# B&R Automation Studio project PloterCNC (part 6)

#### Main.st
```iecst
PROGRAM _INIT
	gParameter;
	UISetup.RecipeListSize	:= 20;
	i; // selected index

END_PROGRAM

PROGRAM _CYCLIC

	// basic settings for recipes
	MpRecipeXml_0(MpLink := ADR(gRecipeXml), Enable := TRUE, DeviceName := ADR('CF'), FileName := ADR('recipe') );

	MpRecipeRegPar_0(MpLink := ADR(gRecipeXml), Enable := TRUE, PVName := ADR('gParameter') );

	MpRecipeUI_0(MpLink := ADR(gRecipeXml), Enable := TRUE, UISetup := UISetup, UIConnect := ADR(UIConnect));

	UIConnect.Recipe.Filter:='*.xml';

	FOR k:=0 TO 4 DO
		memset(ADR(TempLine[k]),0,SIZEOF(TempLine[k]));
		memset(ADR(DataProvider0[k]),0, SIZEOF(DataProvider0[k]));
	END_FOR;

	FOR i:=0 TO 4 DO
		TempLine[0]:='{"value":"';
		TempLine[1]:=INT_TO_STRING(i);
		TempLine[2]:='","text":"';
		TempLine[3]:=UIConnect.Recipe.List.Names[i];
		TempLine[4]:='"}';

		nextAddr:=strcat(ADR(DataProvider0[i]), ADR(TempLine[0]));

		FOR j:=1 TO 4 DO
			strcat(nextAddr,ADR(TempLine[j]));
		END_FOR;

	END_FOR;

	// Messagebox informs that the maximum number of recipes has been reached

	IF UIConnect.Recipe.List.MaxSelection>=5 AND CreatingRecipe  THEN
		gMsgBox4:=TRUE;
		CreatingRecipe := FALSE;
	END_IF;

		END_PROGRAM

PROGRAM _EXIT

	MpRecipeXml_0.Save					:= TRUE;
	MpRecipeXml_0.Enable				:=FALSE;
	MpRecipeXml_0();

	MpRecipeRegPar_0.Enable				:=FALSE;
	MpRecipeRegPar_0();

		END_PROGRAM
```

### Program Logical/RuchZGCode

#### Main.st
```iecst
PROGRAM _INIT
	(* Insert code here *)
	CncName := '';
	CncNameCopy := '';
	toolDown;
	toolUp;
	MC_BR_MFunction_0(AxesGroup :=ADR(gCncXZ) , Enable :=TRUE , MFunction :=50);
	MC_BR_MFunction_1(AxesGroup :=ADR(gCncXZ) , Enable :=TRUE , MFunction :=60);
END_PROGRAM

PROGRAM _CYCLIC

	//Transfering name of the opened file in MotionPad to the initialization of CNC

	IF MpCnc2Axis_0.PowerOn AND MpCnc2Axis_0.IsHomed AND MoveMachine = 1 THEN

	CncNameCopy := DELETE(CncName, 12, 0);
		CncParameters.ProgramName := CncNameCopy;
		MoveMachine := 2;
		IF  strcmp(ADR(CncNameCopy),ADR('')) <> 0 THEN
			MpCnc2Axis_0.MoveProgram := TRUE;
		END_IF

	ELSIF MpCnc2Axis_0.MoveDone THEN
		CncName := '';
		CncNameCopy := '';
		MpCnc2Axis_0.MoveProgram := FALSE;
	END_IF

	//Error control, showing the Error Dialog and reseting errors
	IF MpCnc2Axis_0.Error THEN
		DialogErrorVisible := TRUE;
		MpCnc2Axis_0.Stop := TRUE;
		MpCnc2Axis_0.MoveProgram := FALSE;
	END_IF

	IF MpCnc2Axis_0.Error = FALSE THEN
		MpCnc2Axis_0.ErrorReset := FALSE;
	END_IF

	MC_BR_MFunction_0();
	MC_BR_MFunction_1();
	IF EDGEPOS(toolUp) THEN
		gActiveTool:=FALSE;
		MC_BR_MFunction_0.Reset:=TRUE;
	ELSE
		MC_BR_MFunction_0.Reset:=FALSE;
	END_IF

	IF EDGEPOS(toolDown) THEN
		gActiveTool:=TRUE;
		MC_BR_MFunction_1.Reset:=TRUE;
	ELSE
		MC_BR_MFunction_1.Reset:=FALSE;
	END_IF

END_PROGRAM

PROGRAM _EXIT
	(* Insert code here *)

END_PROGRAM
```

### Package Logical/Sources/Infrastructure - Infrastructure package

### Program Logical/Sources/Infrastructure/SMTP (IEC) - Mail notification via smtp task

#### Smtp.st - Smtp init, cyclic, exit code
```iecst
(*********************************************************************************
 * Copyright:	Bernecker+Rainer
 * Author:		pawlikb
 * Created:		April 23, 2019/8:53 AM
 * Description:
 *			What:	Task handles e-mail notfications about active alarms.
 *			How:	Timer is counting up to INTERVAL_TIME. During this time active
					alarms are registered and then the e-mail with combined information is sent
					and the timer is reset.
 *			Limits:	It is necessary to provide Internet access for the PLC.
					When used with SiteManager the default gateway must be set to DEV IP of the SiteManager,
					and Routing (Scada) Agent must be configured. Please see attached documentation.

 *********************************************************************************)

PROGRAM _INIT
	(* Smtp default configuration *)
	Smtp.Parameters.Host		:=	HOST;
	Smtp.Parameters.User		:=	USER;
	Smtp.Parameters.Password	:=	PASSWORD;
	Smtp.Parameters.Sender		:=	SENDER;
	Smtp.Parameters.Receiver	:=	RECEIVER;
	Smtp.Parameters.Subject		:=	SUBJECT;
	Smtp.Parameters.Text		:=	HEADER;
	Smtp.Parameters.Domain		:=	DOMAIN;				//Usually domain name is not needed
	Smtp.Parameters.Timeout		:=	0;					//If 0 specified then default 120s is used
	Smtp.Parameters.Port		:=	PORT;				//If 0 specified then default port for SMTP (25) is used

	(* Attachment *)
	Smtp.Parameters.AttachmentCnt		:=	0;
	Smtp.Parameters.Attachment.type		:=	smtpATT_TYPE_DATMOD;
	Smtp.Parameters.Attachment.pData	:=	ADR('DatObj');

	(* Timer configuration - get task class cycle time *)
	Smtp.FB.RTInfo.enable	:=	TRUE;
	Smtp.FB.RTInfo();

END_PROGRAM

PROGRAM _CYCLIC

//	(* Increment timer *)
//	Smtp.Status.Timer	:=	Smtp.Status.Timer + Smtp.FB.RTInfo.cycle_time/1000;
//
//	(* Reset timer and send e-mail *)
//	IF Smtp.Status.Timer >= (INTERVAL_TIME * 60) THEN
//		Smtp.Status.Timer	:=	0;
//
//		(* Send email if any alarm was set *)
//		IF Smtp.Status.AlarmActive THEN
////			Smtp.Cmd.Send		:=	TRUE;
////			Smtp.Cmd.SendSSL	:=	TRUE;
//		END_IF;
//	END_IF;
//
//	(* Check for active alarms *)
//	Smtp.Status.AlarmActive	:=	FALSE;
//	FOR i:=0 TO 10 DO
////		Smtp.Status.AlarmActive	:=	Smtp.Status.AlarmActive	OR	[i];
//
//	END_FOR;

	(* Disable function blocks - will be enabled in a state machine *)
	Smtp.FB.SmtpSend.enable		:=	FALSE;
	Smtp.FB.SmtpsSend.enable	:=	FALSE;

	(* State machine *)
	CASE Smtp.Status.State OF

		STATE_SMTP_WAIT:
			(* Command send via SMTP *)
			IF Smtp.Cmd.Send THEN
				(* Prepare message *)
				actText;
				(* Send *)
				Smtp.Status.State	:=	STATE_SMTP_SEND;
			END_IF;

			(* Command send via SMTP with encryption *)
			IF Smtp.Cmd.SendSSL THEN
				(* Prepare message *)
				actText;
				(* Send *)
				Smtp.Status.State	:=	STATE_SMTP_SEND_SSL;
			END_IF;

		STATE_SMTP_SEND:
			(* Enable function block *)
			Smtp.FB.SmtpSend.enable	:=	TRUE;

			(* Assign Mail Parameters *)
			Smtp.FB.SmtpSend.pHost			:=	ADR(Smtp.Parameters.Host);
			Smtp.FB.SmtpSend.pUser			:=	0;	//ADR(Smtp.Parameters.User);
			Smtp.FB.SmtpSend.pPassword		:=	0;	//ADR(Smtp.Parameters.Password);
			Smtp.FB.SmtpSend.pSender		:=	ADR(Smtp.Parameters.Sender);
			Smtp.FB.SmtpSend.pReceiver		:=	ADR(Smtp.Parameters.Receiver);
			Smtp.FB.SmtpSend.pSubject		:=	ADR(Smtp.Parameters.Subject);
			Smtp.FB.SmtpSend.pText			:=	ADR(Smtp.Parameters.Text);
			Smtp.FB.SmtpSend.pDomain		:=	0;	//ADR(Smtp.Parameters.Domain);
			Smtp.FB.SmtpSend.pAttachment	:=	ADR(Smtp.Parameters.Attachment);
			Smtp.FB.SmtpSend.attcnt			:=	Smtp.Parameters.AttachmentCnt;
			Smtp.FB.SmtpSend.timeout		:=	Smtp.Parameters.Timeout;
			Smtp.FB.SmtpSend.port			:=	Smtp.Parameters.Port;

			(* Jump Conditions *)
			IF Smtp.FB.SmtpSend.status = ERR_OK THEN
				Smtp.FB.SmtpSend.enable	:=	FALSE;
				Smtp.Status.State		:=	STATE_SMTP_WAIT;
			ELSIF Smtp.FB.SmtpSend.status = ERR_FUB_BUSY THEN
				(* BUSY *)
			ELSE
				Smtp.Status.State	:=	STATE_SMTP_ERROR;
			END_IF;

		STATE_SMTP_SEND_SSL:
			(* Enable function block *)
			Smtp.FB.SmtpsSend.enable	:=	TRUE;

			(* Assign Mail Parameters *)
			Smtp.FB.SmtpsSend.pHost			:=	ADR(Smtp.Parameters.Host);
			Smtp.FB.SmtpsSend.pUser			:=	ADR(Smtp.Parameters.User);
			Smtp.FB.SmtpsSend.pPassword		:=	ADR(Smtp.Parameters.Password);
			Smtp.FB.SmtpsSend.pSender		:=	ADR(Smtp.Parameters.Sender);
			Smtp.FB.SmtpsSend.pReceiver		:=	ADR(Smtp.Parameters.Receiver);
			Smtp.FB.SmtpsSend.pSubject		:=	ADR(Smtp.Parameters.Subject);
			Smtp.FB.SmtpsSend.pText			:=	ADR(Smtp.Parameters.Text);
			Smtp.FB.SmtpsSend.pDomain		:=	ADR(Smtp.Parameters.Domain);
			Smtp.FB.SmtpsSend.pAttachment	:=	ADR(Smtp.Parameters.Attachment);
			Smtp.FB.SmtpsSend.attcnt		:=	Smtp.Parameters.AttachmentCnt;
			Smtp.FB.SmtpsSend.timeout		:=	Smtp.Parameters.Timeout;
			Smtp.FB.SmtpsSend.port			:=	Smtp.Parameters.Port;
			Smtp.FB.SmtpsSend.sslCfgIdent	:=	0;	//Default SSL Configuration

			(* Jump Conditions *)
			IF Smtp.FB.SmtpsSend.status	= ERR_OK THEN
				Smtp.FB.SmtpsSend.enable	:=	FALSE;
				Smtp.Status.State	:=	STATE_SMTP_WAIT;
			ELSIF Smtp.FB.SmtpsSend.status	=	ERR_FUB_BUSY THEN
				(* BUSY *)
			ELSE
				Smtp.Status.State	:=	STATE_SMTP_ERROR;
			END_IF;

		STATE_SMTP_ERROR:
			(* Auto reset *)
			Smtp.Cmd.ErrorReset	:=	TRUE;

			(* Command error reset *)
			IF Smtp.Cmd.ErrorReset THEN
				Smtp.Status.State	:=	STATE_SMTP_WAIT;
			END_IF;

	END_CASE;

	(* Call Function Blocks *)
	Smtp.FB.SmtpSend();
	Smtp.FB.SmtpsSend();

	(* Reset Commands *)
	IF Smtp.Cmd.Send AND Smtp.Status.State = STATE_SMTP_SEND THEN
		Smtp.Cmd.Send		:=	FALSE;
	END_IF;

	IF Smtp.Cmd.SendSSL AND Smtp.Status.State = STATE_SMTP_SEND_SSL THEN
		Smtp.Cmd.SendSSL	:=	FALSE;
	END_IF;

	IF Smtp.Cmd.ErrorReset AND Smtp.Status.State = STATE_SMTP_WAIT THEN
		Smtp.Cmd.ErrorReset	:=	FALSE;
	END_IF;

END_PROGRAM

PROGRAM _EXIT
	(* Disable function blocks *)
	Smtp.FB.SmtpSend	(enable	:=	FALSE);
	Smtp.FB.SmtpsSend	(enable	:=	FALSE);

END_PROGRAM
```

#### Smtp.typ - Smtp local data types
```iecst
(**** SMTP ****)

TYPE
	SmtpType : 	STRUCT
		Parameters : SmtpParametersType;
		Status : SmtpStatusType;
		Cmd : SmtpCmdType;
		FB : SmtpFBType;
	END_STRUCT;
	SmtpParametersType : 	STRUCT
		Host : STRING[80];
		User : STRING[80];
		Password : STRING[80];
		Sender : STRING[80];
		Receiver : STRING[80];
		Text : STRING[255];
		Subject : STRING[80];
		Attachment : smtpATTACHMENT_typ;
		AttachmentCnt : USINT;
		Domain : STRING[80];
		Timeout : UDINT;
		Port : UINT;
	END_STRUCT;
	SmtpStatusType : 	STRUCT
		State : SmtpStatusStateEnum;
		Timer : UDINT;
		AlarmActive : BOOL;
	END_STRUCT;
	SmtpStatusStateEnum :
		(
		STATE_SMTP_WAIT,
		STATE_SMTP_SEND,
		STATE_SMTP_SEND_SSL,
		STATE_SMTP_ERROR
		);
	SmtpCmdType : 	STRUCT
		SendSSL : BOOL;
		Send : BOOL;
		ErrorReset : BOOL;
	END_STRUCT;
	SmtpFBType : 	STRUCT
		SmtpSend : SmtpSend;
		SmtpsSend : SmtpsSend;
		RTInfo : RTInfo;
	END_STRUCT;
END_TYPE
```

#### Smtp.var - Smtp local variables
```iecst
(**** Constants ****)
VAR CONSTANT
	INTERVAL_TIME : UDINT := 15; (*Interval time in minutes*)
	HOST : STRING[80] := 'smtp.gmail.com'; (*Use plain IP so that DNS is not needed*)
	PORT : UINT := 465; (*SMTP server port*)
	USER : STRING[80] := '0'; (*User of the email account*)
	PASSWORD : STRING[80] := '0'; (*Password*)
	SENDER : STRING[80] := 'lis.weronika.m@gmail.com@gmail.com'; (*Sender*)
	RECEIVER : STRING[80] := 'lis.weronika.m@gmail.com'; (*Receiver*)
	SUBJECT : STRING[80] := 'Hello'; (*Subject of the email*)
	HEADER : STRING[80] := 'Hello World!'; (*Header of the email*)
	FOOTER : STRING[80] := 'This email was sent automatically by SalesCubeKrk. Please do not respond.'; (*Footer of the email*)
	DOMAIN : STRING[80] := 'gmail.com';
END_VAR
(**** SMTP ****)
VAR
	Smtp : SmtpType; (*Smtp structure*)
	i : USINT;
END_VAR
```

#### actText.st - Action preparing text for email
```iecst
(*********************************************************************************
 * Copyright:	Bernecker+Rainer
 * Author:		pawlikb
 * Created:		April 23, 2019/9:41 AM
 * Description:
 *			What:	Action prepares text for the email
 *			How:	Checks if alarm was set, if yes then it appends appropriate message
 *			Limits:
 *********************************************************************************)

ACTION actText:

	(* Header *)
	//Smtp.Parameters.Text	:=	HEADER;

	(* Check and append main text *)

	(* Footer *)
//	brsstrcat(ADR(Smtp.Parameters.Text),ADR(FOOTER));

END_ACTION
```

### Program Logical/Sources/Infrastructure/ICMP (IEC) - Icmp task

#### Icmp.st - Init, cyclic, exit code
```iecst
(*********************************************************************************
 * Copyright:	Bernecker+Rainer
 * Author:		pawlikb
 * Created:		January 8, 2020/3:17 PM
 * Description:
 *			What:	Ping
 *			How:	AsICMP
 *			Limits:
 *********************************************************************************)
PROGRAM _INIT
	(* Default values *)
	Icmp.Parameter.Timeout	:=	DEFAULT_TIMEOUT;

END_PROGRAM

PROGRAM _CYCLIC

	(* State machine *)
	CASE Icmp.Status.State OF

		STATE_ICMP_WAIT:
			(* Command Ping *)
			IF Icmp.Cmd.Ping THEN
				Icmp.Cmd.Ping				:=	FALSE;
				Icmp.FB.IcmpPing.timeout	:=	Icmp.Parameter.Timeout/10;
				Icmp.Status.State			:=	STATE_ICMP_PING;
			END_IF;

		STATE_ICMP_PING:
			(* Configure function block *)
			Icmp.FB.IcmpPing.enable	:=	TRUE;
			Icmp.FB.IcmpPing.pHost	:=	ADR(Icmp.Parameter.Host);

			(* Call function block *)
			Icmp.FB.IcmpPing();

			(* Jump conditions *)
			IF Icmp.FB.IcmpPing.status = ERR_OK THEN
				Icmp.Status.Result			:=	Icmp.FB.IcmpPing.timeout *10;	//1 = 10ms
				Icmp.FB.IcmpPing.timeout	:=	Icmp.FB.IcmpPing.timeout -1;	//Decrease timeout
				Icmp.FB.IcmpPing.enable		:=	FALSE;
				Icmp.Status.State			:=	STATE_ICMP_PING;

				(* Response time < 10ms. If zero is specified default timeout is used = 10ms *)
				IF Icmp.FB.IcmpPing.timeout > Icmp.Parameter.Timeout THEN
					Icmp.Status.Result	:=	10;
					Icmp.Status.State	:=	STATE_ICMP_WAIT;
				END_IF;

			ELSIF Icmp.FB.IcmpPing.status = ERR_FUB_BUSY THEN
				(* BUSY *)

			ELSIF Icmp.FB.IcmpPing.status = icmpERR_NO_RESPONSE THEN
				Icmp.FB.IcmpPing.enable		:=	FALSE;
				Icmp.Status.State			:=	STATE_ICMP_WAIT;

			ELSE
				Icmp.FB.IcmpPing.enable		:=	FALSE;
				Icmp.Status.State			:=	STATE_ICMP_WAIT;
			END_IF;
	END_CASE;

END_PROGRAM

PROGRAM _EXIT
	(* Insert code here *)

END_PROGRAM
```

#### Icmp.typ - Local data types
```iecst
TYPE
	IcmpType : 	STRUCT
		Parameter : IcmpParameterType;
		Cmd : IcmpCmdType;
		Status : IcmpStatusType;
		FB : IcmpFBType;
	END_STRUCT;
	IcmpParameterType : 	STRUCT
		Host : STRING[80];
		Timeout : UINT; (*1 = 10ms*)
	END_STRUCT;
	IcmpCmdType : 	STRUCT
		Ping : BOOL;
	END_STRUCT;
	IcmpStatusType : 	STRUCT
		State : IcmpStatusStateEnum;
		Result : UINT;
	END_STRUCT;
	IcmpStatusStateEnum :
		(
		STATE_ICMP_WAIT,
		STATE_ICMP_PING
		);
	IcmpFBType : 	STRUCT
		IcmpPing : IcmpPing;
	END_STRUCT;
END_TYPE
```

#### Icmp.var - Local variables
```iecst
(**** Constants ****)
VAR CONSTANT
	DEFAULT_TIMEOUT : UINT := 100; (*Ping timeout - 100ms*)
END_VAR
(**** Variables ****)
VAR
	Icmp : IcmpType; (*Icmp structure*)
END_VAR
```

### Program Logical/Sources/Alarm

#### Variables.var
```iecst
VAR
	MpAlarmXHistoryGlobal : MpAlarmXHistory;
	MpAlarmXCoreGeneral : MpAlarmXCore;
	MpAlarmXCoreGlobal : MpAlarmXCore;
	MpAlarmXCoreCnc : MpAlarmXCore;
	MpAlarmXCoreFile : MpAlarmXCore;
END_VAR
```

#### Main.st
```iecst
PROGRAM _INIT

	MpAlarmXCoreGeneral.Enable := TRUE;
	MpAlarmXCoreGeneral.MpLink := ADR(gAlarmXGeneral);

	MpAlarmXCoreFile.Enable := TRUE;
	MpAlarmXCoreFile.MpLink := ADR(gAlarmXFile);

	MpAlarmXCoreCnc.Enable := TRUE;
	MpAlarmXCoreCnc.MpLink := ADR(gAlarmXCnc);

	MpAlarmXCoreGlobal.Enable := TRUE;
	MpAlarmXCoreGlobal.MpLink := ADR(gAlarmXCoreGlobal);

	MpAlarmXHistoryGlobal.Enable := TRUE;
	MpAlarmXHistoryGlobal.MpLink := ADR(gAlarmXHistory);
END_PROGRAM

PROGRAM _CYCLIC

	IF MpAlarmXCoreGlobal.ActiveAlarms>0 OR MpAlarmXCoreGlobal.PendingAlarms>0  THEN
		gAlarmActive:=TRUE;
	ELSE
		gAlarmActive:=FALSE;
	END_IF;

	MpAlarmXCoreGeneral();
	MpAlarmXCoreFile();
	MpAlarmXCoreCnc();
	MpAlarmXCoreGlobal();
	MpAlarmXHistoryGlobal();

END_PROGRAM

PROGRAM _EXIT

	MpAlarmXCoreGlobal.Enable := FALSE;

	MpAlarmXCoreFile.Enable := FALSE;
	MpAlarmXCoreCnc.Enable := FALSE;
	MpAlarmXCoreGeneral.Enable := FALSE;

	MpAlarmXHistoryGlobal.Enable := FALSE;

	MpAlarmXCoreGeneral();
	MpAlarmXCoreFile();
	MpAlarmXCoreCnc();
	MpAlarmXCoreGlobal();
	MpAlarmXHistoryGlobal();

END_PROGRAM
```

### Program Logical/Sources/CNC_Programs/ManualContr

#### Main.st
```iecst
PROGRAM _INIT

	gStartValueChanging;
	MpCnc2Axis_0;
	CncParameters;
	gActiveTool;

	gMoveAbsoluteX:=TRUE;
	gMoveAbsoluteY:=TRUE;

END_PROGRAM

PROGRAM _CYCLIC

	IF gManualContr OR ButtonEnable=FALSE THEN
		gAutomaticContr:=FALSE;
	ELSE
		gAutomaticContr:=TRUE;
	END_IF;

	IF MpCnc2Axis_0.MoveProgram THEN
	  gManualContr:=FALSE;
	END_IF;

	(*When activating manual control*)
	IF EDGEPOS(gManualContr) THEN
	MpBasicParametersX.Position:=MpCnc2Axis_0.X;
	MpBasicParametersY.Position:=MpCnc2Axis_0.Y;
	END_IF

	(*Manual control operating mode switched on with a button in Visu*)
	IF gManualContr THEN

		(*Movement controlled by sliders and text input in visualization*)

		PosX:=LREAL_TO_INT(MpBasicParametersX.Position);
		PosY:=LREAL_TO_INT(MpBasicParametersY.Position);

		IF MpBasicParametersX.Position=INT_TO_LREAL(CncPosX) THEN
			gMoveAbsoluteX:=FALSE;
		END_IF;

		IF MpBasicParametersY.Position=INT_TO_LREAL(CncPosY) THEN
			gMoveAbsoluteY:=FALSE;
		END_IF;

		(*Movement in X (MOVE ABSOLUTE) *)
		IF gMoveAbsoluteX THEN
			MpAxisBasicX.MoveAbsolute:=TRUE;
		END_IF;

		IF MpAxisBasicX.MoveDone=TRUE THEN
			MpAxisBasicX.MoveAbsolute:=FALSE;
			gMoveAbsoluteX:=FALSE;
		END_IF;

		IF EDGENEG(gMoveAbsoluteX) AND CncPosX<>PosX THEN
			gMoveAbsoluteX:=TRUE;
		END_IF;

		(*Movement in Y  (MOVE ABSOLUTE) *)

		IF gMoveAbsoluteY THEN
			MpAxisBasicY.MoveAbsolute:=TRUE;
		END_IF;

		IF MpAxisBasicY.MoveDone=TRUE THEN
			MpAxisBasicY.MoveAbsolute:=FALSE;
			gMoveAbsoluteY:=FALSE;
		END_IF;

		IF EDGENEG(gMoveAbsoluteY) AND CncPosY<>PosY THEN
			gMoveAbsoluteY:=TRUE;
		END_IF;

	ELSIF gManualContr=FALSE THEN
		MpAxisBasicX.MoveAbsolute:=FALSE;
		MpAxisBasicY.MoveAbsolute:=FALSE;
	END_IF;

	(*Movement control with ARROWS in visualization*)

	(*Arrows parameters*)

	MpBasicParametersX.Jog.Velocity:=gParameter.set_X_vel;
	MpBasicParametersY.Jog.Velocity:=gParameter.set_Z_vel;
	MpBasicParametersX.Jog.Acceleration:=gParameter.limit_acc;
	MpBasicParametersY.Jog.Acceleration:=gParameter.limit_acc;
	MpBasicParametersX.Jog.Deceleration:=gParameter.limit_dec;
	MpBasicParametersY.Jog.Deceleration:=gParameter.limit_dec;

	MpBasicParametersX.Jog.LimitPosition.FirstPosition:=0;
	MpBasicParametersX.Jog.LimitPosition.LastPosition:=520;
	MpBasicParametersY.Jog.LimitPosition.FirstPosition:=0;
	MpBasicParametersY.Jog.LimitPosition.LastPosition:=420;

	(*JOG MOVEMENT - NEGATIVE AND POSITIVE*)
	IF MpCnc2Axis_0.MoveActive AND (EDGENEG(MpAxisBasicX.JogNegative) OR EDGENEG(MpAxisBasicY.JogNegative) OR EDGENEG(MpAxisBasicX.JogPositive) OR EDGENEG(MpAxisBasicY.JogPositive)) THEN
	GetThere:=TRUE;
	END_IF;

	IF GetThere THEN
		MpBasicParametersY.Position:=MpCnc2Axis_0.Y;
		MpBasicParametersX.Position:=MpCnc2Axis_0.X;
	END_IF;

	IF MpCnc2Axis_0.MoveActive=FALSE THEN
		GetThere:=FALSE;
	END_IF

	(*Go Up, GoDown, GoLeft and GoRight are variables connected to the arrows in visu*)
	(*UP*)
	IF GoUp=TRUE THEN
		//	MpBasicParametersY.Position:=INT_TO_LREAL(CncPosY);
		MpBasicParametersY.Position:=MpCnc2Axis_0.Y;
		MpAxisBasicY.MoveAbsolute:=FALSE;
		MpAxisBasicY.JogNegative:=TRUE;

	ELSIF GoUp=FALSE THEN
		MpAxisBasicY.JogNegative:=FALSE;
	END_IF;

	(*DOWN*)
	IF GoDown THEN
		MpBasicParametersY.Position:=INT_TO_LREAL(CncPosY);
		MpAxisBasicY.MoveAbsolute:=FALSE;
		MpAxisBasicY.JogPositive:=TRUE;

	ELSIF GoDown=FALSE THEN
		MpAxisBasicY.JogPositive:=FALSE;
	END_IF;

	(*LEFT*)
	IF GoLeft  THEN
		MpBasicParametersX.Position:=INT_TO_LREAL(CncPosX);
		MpAxisBasicX.MoveAbsolute:=FALSE;
		MpAxisBasicX.JogNegative:=TRUE;

	ELSIF GoLeft=FALSE THEN
		MpAxisBasicX.JogNegative:=FALSE;
	END_IF;

		(*RIGHT*)
	IF GoRight THEN
		MpBasicParametersX.Position:=INT_TO_LREAL(CncPosX);
		MpAxisBasicX.MoveAbsolute:=FALSE;
		MpAxisBasicX.JogPositive:=TRUE;

	ELSIF GoRight=FALSE THEN
		MpAxisBasicX.JogPositive:=FALSE;
	END_IF;

	(*Limits for movement in both directions (x,y) *)

	IF MpBasicParametersY.Position>=420 THEN
		MpBasicParametersY.Position:=420;

	ELSIF MpBasicParametersY.Position<=0 THEN
		MpBasicParametersY.Position:=0;
	END_IF;

	IF MpBasicParametersX.Position>=520 THEN
		MpBasicParametersX.Position:=520;

	ELSIF MpBasicParametersX.Position<=0 THEN
		MpBasicParametersX.Position:=0;
	END_IF;

	(* A dot showing the position of the tool*)
	pointString:='<circle cx="';

	pointStrX:=REAL_TO_STRING(CncPosX*1.2);
	pointStrY:=REAL_TO_STRING(CncPosY*1.2);

	strHelp:='" cy="';
	strcat(ADR(pointString),ADR(pointStrX));
	strcat(ADR(pointString),ADR(strHelp));
	strcat(ADR(pointString),ADR(pointStrY));
	strHelp:='" r="5" stroke="black" stroke-width="3" fill="red" />';
	strcat(ADR(pointString),ADR(strHelp));

	MpAxisBasicX();
	MpAxisBasicY();

	IF MpAxisBasicX.Velocity=0 THEN
		gCurrentX:=0;
	ELSIF MpAxisBasicX.Velocity<0 THEN
		gCurrentX:=-MpAxisBasicX.Velocity*0.01+0.48;
	ELSIF MpAxisBasicX.Velocity>0 THEN
		gCurrentX:=MpAxisBasicX.Velocity*0.01+0.48;
		END_IF;

		IF MpAxisBasicY.Velocity=0 THEN
		gCurrentY:=0;
	ELSIF MpAxisBasicY.Velocity<0 THEN
		gCurrentY:=-MpAxisBasicY.Velocity*0.01+0.48;
	ELSIF MpAxisBasicY.Velocity>0 THEN
		gCurrentY:=MpAxisBasicY.Velocity*0.01+0.48;
	END_IF;

VisuAction;

END_PROGRAM

PROGRAM _EXIT

END_PROGRAM
```

#### VisuAction.st
```iecst
ACTION VisuAction:

	Show;
	NumericInput;
	SliderInput;

END_ACTION
```

### Program Logical/Sources/CNC_Programs/RuchZGCode

#### Main.st
```iecst
PROGRAM _INIT
	(* Insert code here *)
	CncName := '';
	CncNameCopy := '';
	toolDown;
	toolUp;
	MC_BR_MFunction_0(AxesGroup :=ADR(gCncXZ) , Enable :=TRUE , MFunction :=50);
	MC_BR_MFunction_1(AxesGroup :=ADR(gCncXZ) , Enable :=TRUE , MFunction :=60);
END_PROGRAM

PROGRAM _CYCLIC

	//Transfering name of the opened file in MotionPad to the initialization of CNC

	IF MpCnc2Axis_0.PowerOn AND MpCnc2Axis_0.IsHomed AND MoveMachine = 1 THEN

	CncNameCopy := DELETE(CncName, 12, 0);
		CncParameters.ProgramName := CncNameCopy;
		MoveMachine := 2;
		IF  strcmp(ADR(CncNameCopy),ADR('')) <> 0 THEN
			MpCnc2Axis_0.MoveProgram := TRUE;
		END_IF

	ELSIF MpCnc2Axis_0.MoveDone THEN
		CncName := '';
		CncNameCopy := '';
		MpCnc2Axis_0.MoveProgram := FALSE;
	END_IF

	//Error control, showing the Error Dialog and reseting errors
	IF MpCnc2Axis_0.Error THEN
		DialogErrorVisible := TRUE;
		MpCnc2Axis_0.Stop := TRUE;
		MpCnc2Axis_0.MoveProgram := FALSE;
	END_IF

	IF MpCnc2Axis_0.Error = FALSE THEN
		MpCnc2Axis_0.ErrorReset := FALSE;
	END_IF

	MC_BR_MFunction_0();
	MC_BR_MFunction_1();
	IF EDGEPOS(toolUp) THEN
		gActiveTool:=FALSE;
		MC_BR_MFunction_0.Reset:=TRUE;
	ELSE
		MC_BR_MFunction_0.Reset:=FALSE;
	END_IF

	IF EDGEPOS(toolDown) THEN
		gActiveTool:=TRUE;
		MC_BR_MFunction_1.Reset:=TRUE;
	ELSE
		MC_BR_MFunction_1.Reset:=FALSE;
	END_IF

END_PROGRAM

PROGRAM _EXIT
	(* Insert code here *)

END_PROGRAM
```

### Program Logical/Sources/live_drawing/live_draw (IEC)

#### Types.typ
```iecst
TYPE
	shape_enum :
		(
		circle,
		line,
		rectangle,
		star,
		arc
		);
END_TYPE
```

#### Main.st
```iecst
PROGRAM _INIT

	readX;
	readY;

END_PROGRAM

PROGRAM _CYCLIC

	(*Warning*)
	IF InfoString='Shape outside drawing field!' THEN
		gMsgBox:=TRUE;
	ELSE
		gMsgBox:=FALSE;
	END_IF;

	IF InfoString='Radius can not be equal to 0!' THEN
		gMsgBox2:=TRUE;
	ELSE
		gMsgBox2:=FALSE;
	END_IF;

	IF InfoString='Distance can not be equal to 0!' THEN
		gMsgBox3:=TRUE;
	ELSE
		gMsgBox3:=FALSE;
	END_IF;

	(*HelpLines*)
	IF HelpLines THEN

		IF (readX-inXlinePosX)<=20 AND (readY-inYlinePosY)<=20 AND (readY-inYlinePosY)>=-20 AND (readX-inXlinePosX)>=-20 THEN
			readX:=REAL_TO_UINT(inXlinePosX);
			readY:=REAL_TO_UINT(inYlinePosY);
		END_IF;

	END_IF;

	CASE curShape OF

		circle:

			CurrentShape:='circle';
			(*-circle drawing-*)
			CASE stage OF
				0:
			InfoString:='Point centre of the circle';
					IF EDGEPOS(cmdDraw) THEN
						cmdDraw:=FALSE;
						RotationAngle:=0;
						strRot:=REAL_TO_STRING(RotationAngle);
						shapeString:='<circle cx="';
						prevReadX:=readX;
						prevReadY:=readY;
						strX:=UINT_TO_STRING(readX);
						strY:=UINT_TO_STRING(readY);

						strHelp:='" cy="';
						strcat(ADR(shapeString),ADR(strX));
						strcat(ADR(shapeString),ADR(strHelp));
						strcat(ADR(shapeString),ADR(strY));
						strHelp:='" r="';
						strcat(ADR(shapeString),ADR(strHelp));
						stage:=1;

						IF prevReadX-CircleRadius<0 OR prevReadY-CircleRadius<0 OR prevReadX+CircleRadius>780 OR prevReadY+CircleRadius>630 THEN
							stage:=1;
						ELSIF CircleRadius=0 THEN
							stage:=2;
						ELSE
							strRadius:=REAL_TO_STRING(CircleRadius);
							strcat(ADR(shapeString),ADR(strRadius));
							strHelp:='" stroke="black" fill="none" />';
							strcat(ADR(shapeString),ADR(strHelp));

							svgStringArray[svgStringArrayIndex]:=shapeString;
							svgStringArrayIndex:=svgStringArrayIndex+1;

							IF svgStringArray[3]<>'' THEN

								(*PositionArray*)
								strHelp:='type:';
								strcat(ADR(PositionString), ADR(strHelp));
								strcat(ADR(PositionString), ADR(CurrentShape));
								strHelp:='; x=';
								strcat(ADR(PositionString), ADR(strHelp));

								strcat(ADR(PositionString), ADR(strX));
								strHelp:='; y=';
								strcat(ADR(PositionString), ADR(strHelp));
								strcat(ADR(PositionString), ADR(strY));;
								strHelp:='; rot=';
								strcat(ADR(PositionString), ADR(strHelp));
								strcat(ADR(PositionString), ADR(strRot));
								strHelp:='';
								strcat(ADR(PositionString), ADR(strHelp));

								PositionArray[PositionArrayIndex]:=PositionString;
								PositionArrayIndex:=PositionArrayIndex+1;
								PositionString:='';

							END_IF;

							stage:=0;

						END_IF;
					END_IF;

				1:
					InfoString:='Shape outside drawing field!';

					IF EDGEPOS(cmdDraw) THEN
						cmdDraw:=FALSE;
						stage:=0;
					END_IF;

				2:
					InfoString:='Radius can not be equal to 0!';
					IF EDGEPOS(cmdDraw) THEN
						cmdDraw:=FALSE;
						stage:=0;
					END_IF;

			END_CASE;

			(*---------------*)
		line:
			(*-line drawing-*)
			CASE stage OF

				0:
					CurrentShape:='line';

					InfoString:='Point first-point of the line';
					IF EDGEPOS(cmdDraw) THEN
						cmdDraw:=FALSE;
						shapeString:='<polyline points="';
						prevReadX:=readX;
						prevReadY:=readY;

						stage:=1;
					END_IF;

				1:
			InfoString:='Point end-point of the line';
					IF EDGEPOS(cmdDraw) THEN
						cmdDraw:=FALSE;
						strPrevX:=UINT_TO_STRING(prevReadX);
						strPrevY:=UINT_TO_STRING(prevReadY);
						strX:=UINT_TO_STRING(readX);
						strY:=UINT_TO_STRING(readY);
						strHelp:=',';
						strcat(ADR(shapeString),ADR(strPrevX));
						strcat(ADR(shapeString),ADR(strHelp));
						strcat(ADR(shapeString),ADR(strPrevY));
						strHelp:=' ';
						strcat(ADR(shapeString),ADR(strHelp));
						strHelp:=',';
						strcat(ADR(shapeString),ADR(strX));
						strcat(ADR(shapeString),ADR(strHelp));
						strcat(ADR(shapeString),ADR(strY));

						strHelp:='" fill="none" stroke="black" />';
						strcat(ADR(shapeString),ADR(strHelp));
						svgStringArray[svgStringArrayIndex]:=shapeString;

						svgStringArrayIndex:=svgStringArrayIndex+1;

						stage:=0;
					END_IF;

			END_CASE;

		(*---------------*)

		rectangle:
			(*-rectangle drawing-*)
			CurrentShape:='rectangle';
			CASE stage OF
				0:
			InfoString:='Point top-left corner of the rectangle';
					IF EDGEPOS(cmdDraw) THEN
						cmdDraw:=FALSE;
						shapeString:='<polyline points="';
						prevReadX:=readX;
						prevReadY:=readY;
						strPrevReadX:=UINT_TO_STRING(prevReadX);
						strPrevReadY:=UINT_TO_STRING(prevReadY);
						strRot:=REAL_TO_STRING(RotationAngle);

						IF prevReadX+readXRec>780 OR prevReadY+readYRec>630 THEN
							cmdDraw:=FALSE;
							stage:=1;
						ELSIF readXRec=0 OR readYRec=0 THEN
							stage:=2;
						ELSE
							strPrevX:=UINT_TO_STRING(prevReadX);
							strPrevY:=UINT_TO_STRING(prevReadY);
							strXRec:=UINT_TO_STRING(prevReadX+readXRec);
							strYRec:=UINT_TO_STRING(prevReadY+readYRec);
							strHelp:=',';
							strcat(ADR(shapeString),ADR(strPrevX));
							strcat(ADR(shapeString),ADR(strHelp));
							strcat(ADR(shapeString),ADR(strPrevY));
							strHelp:=' ';
							strcat(ADR(shapeString),ADR(strHelp));
							strHelp:=',';
							strcat(ADR(shapeString),ADR(strXRec));
							strcat(ADR(shapeString),ADR(strHelp));
							strcat(ADR(shapeString),ADR(strPrevY));
							strHelp:=' ';
							strcat(ADR(shapeString),ADR(strHelp));
							strHelp:=',';
							strcat(ADR(shapeString),ADR(strXRec));
							strcat(ADR(shapeString),ADR(strHelp));
							strcat(ADR(shapeString),ADR(strYRec));
							strHelp:=' ';
							strcat(ADR(shapeString),ADR(strHelp));
							strHelp:=',';
							strcat(ADR(shapeString),ADR(strPrevX));
							strcat(ADR(shapeString),ADR(strHelp));
							strcat(ADR(shapeString),ADR(strYRec));

							strHelp:=' ';
							strcat(ADR(shapeString),ADR(strHelp));
							strHelp:=',';
							strcat(ADR(shapeString),ADR(strPrevX));
							strcat(ADR(shapeString),ADR(strHelp));
							strcat(ADR(shapeString),ADR(strPrevY));
							strHelp:='" transform="rotate(';
							strcat(ADR(shapeString),ADR(strHelp));
							strcat(ADR(shapeString),ADR(strRot));
							strHelp:=' ';
							strcat(ADR(shapeString),ADR(strHelp));
							strcat(ADR(shapeString),ADR(strPrevX));
							strHelp:=',';
							strcat(ADR(shapeString),ADR(strHelp));
							strcat(ADR(shapeString),ADR(strPrevY));
							strHelp:=')"';
							strcat(ADR(shapeString),ADR(strHelp));
							strHelp:=' fill="none" stroke="black" />';
							strcat(ADR(shapeString),ADR(strHelp));
							svgStringArray[svgStringArrayIndex]:=shapeString;

							svgStringArrayIndex:=svgStringArrayIndex+1;

							IF svgStringArray[3]<>'' THEN

								(*PositionArray*)
								strHelp:='type:';
								strcat(ADR(PositionString), ADR(strHelp));
								strcat(ADR(PositionString), ADR(CurrentShape));
								strHelp:='; x=';
								strcat(ADR(PositionString), ADR(strHelp));
								strcat(ADR(PositionString), ADR(strPrevReadX));
								strHelp:='; y=';
								strcat(ADR(PositionString), ADR(strHelp));
								strcat(ADR(PositionString), ADR(strPrevReadY));
								strHelp:='; rot=';
								strcat(ADR(PositionString), ADR(strHelp));
								strcat(ADR(PositionString), ADR(strRot));
								strHelp:='';
								strcat(ADR(PositionString), ADR(strHelp));

								PositionArray[PositionArrayIndex]:=PositionString;
								PositionArrayIndex:=PositionArrayIndex+1;
								PositionString:='';
							END_IF;

							stage:=0;
						END_IF;
					END_IF;

				1:
					InfoString:='Shape outside drawing field!';

					IF EDGEPOS(cmdDraw) THEN
						cmdDraw:=FALSE;
						stage:=0;
					END_IF;

				2:
					InfoString:='Distance can not be equal to 0!';

					IF EDGEPOS(cmdDraw) THEN
						cmdDraw:=FALSE;
						stage:=0;
					END_IF;

			END_CASE;

		(*---------------*)

		star:
			(*-star drawing-*)
			CASE stage OF

				0:
					CurrentShape:='star';
					InfoString:='Point centre of the star';
					strRot:=REAL_TO_STRING(RotationAngle);

					IF EDGEPOS(cmdDraw) THEN
						cmdDraw:=FALSE;
						shapeString:='<polyline points="';
						prevReadX:=readX;
						prevReadY:=readY;
						strPrevReadX:=REAL_TO_STRING(prevReadX);
						strPrevReadY:=REAL_TO_STRING(prevReadY);
						cmdDraw:=FALSE;

						IF prevReadX-radius<0 OR prevReadY-radius<0 OR prevReadX+radius>780 OR prevReadY+radius>630 THEN
							stage:=1;
						ELSIF radius=0 THEN
							stage:=2;
						ELSE
							smallRadius:=radius/3;
							angle:=-18; // degrees
							FOR i:=1 TO 5 DO

								x:=radius*COS(angle/180*PI);
								y:=radius*SIN(angle/180*PI);
								strX:=REAL_TO_STRING(x+prevReadX);
								strY:=REAL_TO_STRING(y+prevReadY);
								strHelp:=',';
								strcat(ADR(shapeString),ADR(strX));
								strcat(ADR(shapeString),ADR(strHelp));
								strcat(ADR(shapeString),ADR(strY));
								strHelp:=' ';
								strcat(ADR(shapeString),ADR(strHelp));

								x:=smallRadius*COS((angle+36)/180*PI);
								y:=smallRadius*SIN((angle+36)/180*PI);

								strX:=REAL_TO_STRING(x+prevReadX);
								strY:=REAL_TO_STRING(y+prevReadY);
								strHelp:=',';
								strcat(ADR(shapeString),ADR(strX));
								strcat(ADR(shapeString),ADR(strHelp));
								strcat(ADR(shapeString),ADR(strY));
								strHelp:=' ';
								strcat(ADR(shapeString),ADR(strHelp));
								angle:=angle+72;

							END_FOR;

							x:=radius*COS(angle/180*PI);
							y:=radius*SIN(angle/180*PI);
							strX:=REAL_TO_STRING(x+prevReadX);
							strY:=REAL_TO_STRING(y+prevReadY);
							strHelp:=',';
							strcat(ADR(shapeString),ADR(strX));
							strcat(ADR(shapeString),ADR(strHelp));
							strcat(ADR(shapeString),ADR(strY));

							strHelp:='" transform="rotate(';
							strcat(ADR(shapeString),ADR(strHelp));
							strcat(ADR(shapeString),ADR(strRot));
							strHelp:=' ';
							strcat(ADR(shapeString),ADR(strHelp));
							strcat(ADR(shapeString),ADR(strPrevReadX));
							strHelp:=',';
							strcat(ADR(shapeString),ADR(strHelp));
							strcat(ADR(shapeString),ADR(strPrevReadY));
							strHelp:=')"';
							strcat(ADR(shapeString),ADR(strHelp));

							strHelp:='" fill="none" stroke="black" />';
							strcat(ADR(shapeString),ADR(strHelp));
							svgStringArray[svgStringArrayIndex]:=shapeString;

							svgStringArrayIndex:=svgStringArrayIndex+1;

							IF svgStringArray[3]<>'' THEN

								(*PositionArray*)
								strHelp:='type:';
								strcat(ADR(PositionString), ADR(strHelp));
								strcat(ADR(PositionString), ADR(CurrentShape));
								strHelp:='; x=';
								strcat(ADR(PositionString), ADR(strHelp));
								strcat(ADR(PositionString), ADR(strPrevReadX));
								strHelp:='; y=';
								strcat(ADR(PositionString), ADR(strHelp));
								strcat(ADR(PositionString), ADR(strPrevReadY));
								strHelp:='; rot=';
								strcat(ADR(PositionString), ADR(strHelp));
								strcat(ADR(PositionString), ADR(strRot));
								strHelp:='';
								strcat(ADR(PositionString), ADR(strHelp));

								PositionArray[PositionArrayIndex]:=PositionString;
								PositionArrayIndex:=PositionArrayIndex+1;
								PositionString:='';
							END_IF;

							stage:=0;
						END_IF;

					END_IF;
				1:
					InfoString:='Shape outside drawing field!';
					IF EDGEPOS(cmdDraw) THEN
						cmdDraw:=FALSE;
						stage:=0;
					END_IF

				2:
					InfoString:='Distance can not be equal to 0!';
					IF EDGEPOS(cmdDraw) THEN
						cmdDraw:=FALSE;
						stage:=0;
					END_IF;

			END_CASE;

	END_CASE;

(*----clearing paper-----*)
	IF EDGEPOS(cmdClear) THEN
		cmdClear:=FALSE;
		FOR i:=3 TO svgStringArrayIndex DO
			svgStringArray[i]:='';
		END_FOR;
		svgStringArrayIndex:=3;
		FOR i:=0 TO PositionArrayIndex DO
			PositionArray[i]:='';
		END_FOR;
		PositionArrayIndex:=0;
	END_IF;
(*------Undo--------*)
	IF EDGEPOS(cmdBack) THEN
		cmdBack:=FALSE;
		IF svgStringArrayIndex>0 THEN
			svgStringArrayIndex:=svgStringArrayIndex-1;
		END_IF
			svgStringArray[svgStringArrayIndex]:='';

		IF PositionArrayIndex>0 THEN
			PositionArrayIndex:=svgStringArrayIndex-1;
		END_IF
		PositionArray[PositionArrayIndex]:='';
	END_IF;

	IF HelpLines THEN

	(* A line showing the position in X*)
	inXlinePosYStr:=REAL_TO_STRING(inXlinePosY);
	inXlinePosXStr:=REAL_TO_STRING(inXlinePosX);
	inXlinePosYStr1:=REAL_TO_STRING(inXlinePosY1);

	svgStringArray[0]:='<polyline points="';
	inXlinePosY1:=0;
	strcat(ADR(svgStringArray[0]),ADR(inXlinePosXStr));
	strHelp:=',';
	strcat(ADR(svgStringArray[0]),ADR(strHelp));
	strcat(ADR(svgStringArray[0]),ADR(inXlinePosYStr1));
	strHelp:=' ';
	strcat(ADR(svgStringArray[0]),ADR(strHelp));
	inXlinePosY:=630;
	strcat(ADR(svgStringArray[0]),ADR(inXlinePosXStr));
	strHelp:=',';
	strcat(ADR(svgStringArray[0]),ADR(strHelp));
	strcat(ADR(svgStringArray[0]),ADR(inXlinePosYStr));
	strHelp:='" fill="none" stroke="red" />';
	strcat(ADR(svgStringArray[0]),ADR(strHelp));

	(* A line showing the position in Y*)
	inYlinePosYStr:=REAL_TO_STRING(inYlinePosY);
	inYlinePosXStr:=REAL_TO_STRING(inYlinePosX);
	inYlinePosXStr1:=REAL_TO_STRING(inYlinePosX1);

	svgStringArray[1]:='<polyline points="';
	inYlinePosX1:=0;
	strcat(ADR(svgStringArray[1]),ADR(inYlinePosXStr1));
	strHelp:=',';
	strcat(ADR(svgStringArray[1]),ADR(strHelp));
	strcat(ADR(svgStringArray[1]),ADR(inYlinePosYStr));
	strHelp:=' ';
	strcat(ADR(svgStringArray[1]),ADR(strHelp));
	inYlinePosX:=780;
	strcat(ADR(svgStringArray[1]),ADR(inYlinePosXStr));
	strHelp:=',';
	strcat(ADR(svgStringArray[1]),ADR(strHelp));
	strcat(ADR(svgStringArray[1]),ADR(inYlinePosYStr));
	strHelp:='" fill="none" stroke="red" />';
	strcat(ADR(svgStringArray[1]),ADR(strHelp));

		(* A circle*)

		svgStringArray[2]:='<circle cx="';

		strHelp:='" cy="';
		strcat(ADR(svgStringArray[2]),ADR(inXlinePosXStr));
		strcat(ADR(svgStringArray[2]),ADR(strHelp));
		strcat(ADR(svgStringArray[2]),ADR(inYlinePosYStr));
		strHelp:='" r="20" stroke="red" stroke-width="1" fill="none" />';
		strcat(ADR(svgStringArray[2]),ADR(strHelp));
	ELSE
		(* A line showing the position in X*)
		inXlinePosYStr:=REAL_TO_STRING(inXlinePosY);
		inXlinePosXStr:=REAL_TO_STRING(inXlinePosX);
		inXlinePosYStr1:=REAL_TO_STRING(inXlinePosY1);

		svgStringArray[0]:='<polyline points="';
		inXlinePosY1:=0;
		strcat(ADR(svgStringArray[0]),ADR(inXlinePosXStr));
		strHelp:=',';
		strcat(ADR(svgStringArray[0]),ADR(strHelp));
		strcat(ADR(svgStringArray[0]),ADR(inXlinePosYStr1));
		strHelp:=' ';
		strcat(ADR(svgStringArray[0]),ADR(strHelp));
		inXlinePosY:=630;
		strcat(ADR(svgStringArray[0]),ADR(inXlinePosXStr));
		strHelp:=',';
		strcat(ADR(svgStringArray[0]),ADR(strHelp));
		strcat(ADR(svgStringArray[0]),ADR(inXlinePosYStr));
		strHelp:='" fill="none" stroke="white" />';
		strcat(ADR(svgStringArray[0]),ADR(strHelp));

		(* A line showing the position in Y*)
		inYlinePosYStr:=REAL_TO_STRING(inYlinePosY);
		inYlinePosXStr:=REAL_TO_STRING(inYlinePosX);
		inYlinePosXStr1:=REAL_TO_STRING(inYlinePosX1);

		svgStringArray[1]:='<polyline points="';
		inYlinePosX1:=0;
		strcat(ADR(svgStringArray[1]),ADR(inYlinePosXStr1));
		strHelp:=',';
		strcat(ADR(svgStringArray[1]),ADR(strHelp));
		strcat(ADR(svgStringArray[1]),ADR(inYlinePosYStr));
		strHelp:=' ';
		strcat(ADR(svgStringArray[1]),ADR(strHelp));
		inYlinePosX:=780;
		strcat(ADR(svgStringArray[1]),ADR(inYlinePosXStr));
		strHelp:=',';
		strcat(ADR(svgStringArray[1]),ADR(strHelp));
		strcat(ADR(svgStringArray[1]),ADR(inYlinePosYStr));
		strHelp:='" fill="none" stroke="white" />';
		strcat(ADR(svgStringArray[1]),ADR(strHelp));

		(* A circle*)

		svgStringArray[2]:='<circle cx="';

		strHelp:='" cy="';
		strcat(ADR(svgStringArray[2]),ADR(inXlinePosXStr));
		strcat(ADR(svgStringArray[2]),ADR(strHelp));
		strcat(ADR(svgStringArray[2]),ADR(inYlinePosYStr));
		strHelp:='" r="20" stroke="white" stroke-width="2" fill="none" />';
		strcat(ADR(svgStringArray[2]),ADR(strHelp));
	END_IF;

	(*------Pass to global---------*)
	gSvgStringArray:=svgStringArray;
	gSvgStringArrayIndex:=svgStringArrayIndex;

END_PROGRAM

PROGRAM _EXIT
	(* Insert code here *)

END_PROGRAM
```

### svgArray.var
```iecst
VAR
	gSvgStringArray : ARRAY[0..999] OF STRING[500];
	gSvgStringArrayIndex : UINT;
END_VAR
```

### Program Logical/UserManagement/UsrMgmtP (IEC)

#### Main.st - Init, cyclic, exit code
```iecst
PROGRAM _INIT

	MpUserXLogin_0.Enable := 1;
	MpUserXLogin_0.MpLink := ADR(gUserXLogin);

	MpUserXManagerUI_0.Enable := 1;
	MpUserXManagerUI_0.MpLink := ADR(gUserXLogin);
	MpUserXManagerUI_0.UIConnect := ADR(MpUserXMgrUIConnect_0);
	MpUserXManagerUI_0.UISetup := MpUserXMgrUISetup_0;

	MpUserXLoginUI_0.Enable := 1;
	MpUserXLoginUI_0.MpLink := ADR(gUserXLogin);
	MpUserXLoginUI_0.UIConnect := ADR(MpUserXLoginUIConnect0);

END_PROGRAM

PROGRAM _CYCLIC

	//DISPLAY SELECTED USER
	SelectedUser := MpUserXMgrUIConnect_0.User.List.UserNames[MpUserXMgrUIConnect_0.User.List.SelectedIndex];

	//DEFAULT DISPLAY ANONYMOUS
	IF MpUserXLoginUIConnect0.CurrentUser = "" THEN
		LoggedAs := "Anonymous";
	ELSE
		LoggedAs := MpUserXLoginUIConnect0.CurrentUser;
	END_IF;

	//ENABLING BUTTONS USER MENU
	IF MpUserXLoginUIConnect0.UserLevel = 100 THEN
		IF SelectedUser = "Administrator" OR SelectedUser = "Anonymous" OR SelectedUser = "Operator" THEN
			RemoveButtonEnabled := 0;
			EditButtonEnabled := 0;
			NewUserButtonEnabled := 1;
		ELSE
			EditButtonEnabled := 1;
			RemoveButtonEnabled := 1;
			NewUserButtonEnabled := 1;
		END_IF;

	ELSIF MpUserXLoginUIConnect0.UserLevel = 50 THEN
		EditButtonEnabled := 0;
		RemoveButtonEnabled := 0;
		NewUserButtonEnabled := 1;
	ELSE
		EditButtonEnabled := 0;
		RemoveButtonEnabled := 0;
		NewUserButtonEnabled := 0;
	END_IF;

	//ENABLING BUTTONS MOREEE
	IF MpUserXLoginUIConnect0.UserLevel = 100 THEN
		Enable.ButonOpenExplorer := 1;
		Enable.ButtonAcknowledge := 1;
		Enable.ButtonAcknowledgeAll := 1;
		Enable.ButtonActivateTool := 1;
		Enable.ButtonConvert := 1;
		Enable.ButtonLoad := 1;
		Enable.ButtonRefresh := 1;
		Enable.ButtonResetErrors := 1;
		Enable.ButtonSave := 1;
		Enable.ButtonSaveGcode := 1;
		Enable.ButtonSaveGcodeAs := 1;
		Enable.ButtonStart := 1;
		Enable.ButtonTurnOff := 1;
		Enable.SetAcc := 1;
		Enable.SetDec := 1;
		Enable.SetVelocityLimit := 1;
		Enable.SetXPos := 1;
		Enable.SetXVelocity := 1;
		Enable.SetYPos := 1;
		Enable.SetYVelocity := 1;
		Enable.ButtonCreate := 1;
		Enable.TextInputCreate := 1;
		Enable.ButtonDelete := 1;

	ELSIF MpUserXLoginUIConnect0.UserLevel = 50 THEN
		Enable.ButonOpenExplorer := 1;
		Enable.ButtonAcknowledge := 1;
		Enable.ButtonAcknowledgeAll := 1;
		Enable.ButtonActivateTool := 1;
		Enable.ButtonConvert := 1;
		Enable.ButtonLoad := 1;
		Enable.ButtonRefresh := 1;
		Enable.ButtonResetErrors := 1;
		Enable.ButtonSave := 1;
		Enable.ButtonSaveGcode := 1;
		Enable.ButtonSaveGcodeAs := 1;
		Enable.ButtonStart := 1;
		Enable.ButtonTurnOff := 1;
		Enable.SetAcc := 1;
		Enable.SetDec := 1;
		Enable.SetVelocityLimit := 0;
		Enable.SetXPos := 0;
		Enable.SetXVelocity := 1;
		Enable.SetYPos := 0;
		Enable.SetYVelocity := 1;
		Enable.ButtonCreate := 1;
		Enable.TextInputCreate := 1;
		Enable.ButtonDelete := 1;
	ELSE
		Enable.ButonOpenExplorer := 0;
		Enable.ButtonAcknowledge := 0;
		Enable.ButtonAcknowledgeAll := 0;
		Enable.ButtonActivateTool := 0;
		Enable.ButtonConvert := 0;
		Enable.ButtonLoad := 0;
		Enable.ButtonRefresh := 0;
		Enable.ButtonResetErrors := 0;
		Enable.ButtonSave := 0;
		Enable.ButtonSaveGcode := 0;
		Enable.ButtonSaveGcodeAs := 0;
		Enable.ButtonStart := 0;
		Enable.ButtonTurnOff := 0;
		Enable.SetAcc := 0;
		Enable.SetDec := 0;
		Enable.SetVelocityLimit := 0;
		Enable.SetXPos := 0;
		Enable.SetXVelocity := 0;
		Enable.SetYPos := 0;
		Enable.SetYVelocity := 0;
		Enable.ButtonCreate := 0;
		Enable.TextInputCreate := 0;
		Enable.ButtonDelete := 0;
	END_IF;

	//DISPALYING FIRST LOGIN DATE OR NO FIRST LOGIN LABEL
	IF MpUserXMgrUIConnect_0.User.Info.FirstLogin = DT#1970-01-01-00:00:00 THEN
		LabelFirstLoginVisible := 1;
		DateFirstLoginVisible := 0;
	ELSE
		LabelFirstLoginVisible := 0;
		DateFirstLoginVisible := 1;
	END_IF;

	//ENABLING LOGIN BUTTON
	IF MpUserXLoginUIConnect0.Login.UserName = "" OR MpUserXLoginUIConnect0.Login.Password = "" THEN
		LoginButtonEnabled := 0;
	ELSE
		LoginButtonEnabled := 1;
	END_IF;

	//DISABLING LOGOUT BUTTON IF NOT LOGGED IN
	IF MpUserXLoginUIConnect0.LoggedIn = 0 THEN
		LogoutButtonEnabled := 0;
	ELSE
		LogoutButtonEnabled := 1;
	END_IF;

	//NEW USER DIALOG ENABLING CONFIRM BUTTON
	IF (MpUserXMgrUIConnect_0.User.Create.Dialog.ConfirmPasswordOk = 1 AND MpUserXMgrUIConnect_0.User.Create.Dialog.UserNameOk = 1) THEN
		DialogNewUserConfirmEnabled := 1;
	ELSE
		DialogNewUserConfirmEnabled := 0;
	END_IF;

	//EDIT USER DIALOG ENABLING CONFIRM BUTTON
	IF (MpUserXMgrUIConnect_0.User.Edit.Dialog.ConfirmPasswordOk = 1 ) THEN
		DialogEditUserConfirmEnabled := 1;
	ELSE
		DialogEditUserConfirmEnabled := 0;
	END_IF;

	//DIALOG NEW USER DISPALY PASSWORD HINT
	IF MpUserXMgrUIConnect_0.User.Create.Dialog.CriteriaNotMet = mpUSERX_PASSWORD_CRIT_NONE THEN
		NewUserPasswordHint := "Password ok";
	ELSIF MpUserXMgrUIConnect_0.User.Create.Dialog.CriteriaNotMet = mpUSERX_PASSWORD_CRIT_LENGTH THEN
		NewUserPasswordHint := "Password too short";
	END_IF;

	//DIALOG NEW USER DISPLAY PASSWORDS MATCH INFO
	IF MpUserXMgrUIConnect_0.User.Create.Dialog.NewPasswordOk = 1 AND MpUserXMgrUIConnect_0.User.Create.Dialog.ConfirmPasswordOk = 1 THEN
		NewUserPasswordOk := "Passwords match";
	ELSE
		NewUserPasswordOk := "Passwords do not match";
	END_IF;

	//USER GROUPS DISPLAY
	CASE MpUserXMgrUIConnect_0.User.Info.Roles[0] OF
		1:
			SelectedUserGroup := "Administrator";
		2:
			SelectedUserGroup := "Anonymous";
		3:
			SelectedUserGroup := "Operator";
	END_CASE;

	//NEW USER ROLE
	MpUserXMgrUIConnect_0.User.Create.Dialog.Roles[0] := NewUserRoleIndex + 2;

	//EDITING USER ROLE
	MpUserXMgrUIConnect_0.User.Edit.Dialog.Roles[0] := EditUserRoleIndex + 2;

	//DIALOG EDIT USER DISPLAY PASSWORD HINT
	IF MpUserXMgrUIConnect_0.User.Edit.Dialog.CriteriaNotMet = mpUSERX_PASSWORD_CRIT_NONE THEN
		EditUserPasswordHint := "Password ok";
	ELSIF MpUserXMgrUIConnect_0.User.Edit.Dialog.CriteriaNotMet = mpUSERX_PASSWORD_CRIT_LENGTH THEN
		EditUserPasswordHint := "Password too short";
	END_IF;

	//DIALOG EDIT USER DISPLAY PASSWORDS MATCH INFO
	IF MpUserXMgrUIConnect_0.User.Edit.Dialog.NewPasswordOk = 1 AND MpUserXMgrUIConnect_0.User.Edit.Dialog.ConfirmPasswordOk = 1 THEN
		EditUserPasswordOk := "Passwords match";
	ELSE
		EditUserPasswordOk := "Passwords do not match";
	END_IF;

	//ERRORS
	IF MpUserXLoginUIConnect0.MessageBox.ErrorNumber = 28673 THEN
		StringError := "User does not exist.";
	ELSIF MpUserXLoginUIConnect0.MessageBox.ErrorNumber = 28672 THEN
		StringError := "Password incorrect.";
	ELSE
		StringError := "No errors?";
	END_IF;

	//FUNCTION CALL
	MpUserXLogin_0();
	MpUserXLoginUI_0();
	MpUserXManagerUI_0();

END_PROGRAM

PROGRAM _EXIT

	MpUserXLogin_0.Enable := 0;
	MpUserXLogin_0();

	MpUserXLoginUI_0.Enable := 0;
	MpUserXLoginUI_0();

	MpUserXManagerUI_0.Enable := 0;
	MpUserXManagerUI_0();

END_PROGRAM
```

#### Variables.var - Local variables
```iecst
VAR
	Enable : EnableType;
	LabelFirstLoginVisible : BOOL;
	DateFirstLoginVisible : BOOL;
	StringError : WSTRING[80];
	EditUserRoleIndex : USINT;
	NewUserRoleIndex : USINT;
	DialogEditUserConfirmEnabled : BOOL;
	DialogNewUserConfirmEnabled : BOOL;
	NewUserButtonEnabled : BOOL;
	EditButtonEnabled : BOOL;
	RemoveButtonEnabled : BOOL;
	LoginButtonEnabled : BOOL;
	LogoutButtonEnabled : BOOL;
	SelectedUser : WSTRING[80];
	EditUserPasswordOk : WSTRING[80];
	NewUserPasswordOk : WSTRING[80];
	SelectedUserGroup : WSTRING[80];
	LoggedAs : WSTRING[80];
	EditUserPasswordHint : WSTRING[80];
	NewUserPasswordHint : WSTRING[80];
	MpUserXLoginUIConnect0 : MpUserXLoginUIConnectType;
	MpUserXLoginUI_0 : MpUserXLoginUI;
	MpUserXLogin_0 : MpUserXLogin;
	MpUserXManagerUI_0 : MpUserXManagerUI;
	MpUserXMgrUIConnect_0 : MpUserXMgrUIConnectType;
	MpUserXMgrUISetup_0 : MpUserXMgrUISetupType;
END_VAR
```

#### Types.typ - Local data types
```iecst
TYPE
	EnableType : 	STRUCT
		ButtonStart : BOOL;
		ButtonResetErrors : BOOL;
		ButtonTurnOff : {REDUND_UNREPLICABLE} BOOL;
		ButtonActivateTool : BOOL;
		ButtonConvert : BOOL;
		ButonOpenExplorer : BOOL;
		ButtonSaveGcode : BOOL;
		ButtonSaveGcodeAs : BOOL;
		ButtonLoad : BOOL;
		ButtonSave : BOOL;
		ButtonRefresh : BOOL;
		SetXPos : BOOL;
		SetYPos : BOOL;
		SetAcc : BOOL;
		SetDec : BOOL;
		SetXVelocity : BOOL;
		SetYVelocity : BOOL;
		SetVelocityLimit : BOOL;
		ButtonAcknowledge : BOOL;
		ButtonAcknowledgeAll : BOOL;
		ButtonDelete : BOOL;
		ButtonCreate : BOOL;
		TextInputCreate : BOOL;
	END_STRUCT;
END_TYPE
```

### Program Logical/UserVisu

#### Variables.var
```iecst
VAR
	Show : BOOL;
	NumericInput : USINT;
	SliderInput : USINT;
END_VAR
```

#### Main.st
```iecst
PROGRAM _INIT

	Show:=FALSE;
	NumericInput:=0;
	SliderInput:=0;

END_PROGRAM

PROGRAM _CYCLIC

END_PROGRAM

PROGRAM _EXIT
	(* Insert code here *)

END_PROGRAM
```

Listed in the project but not available here: Logical/MSpltrFmu/MSpltrLib/Constants.var, Logical/MSpltrFmu/MSpltrLib/fmi2FunctionTypes.h, Logical/MSpltrFmu/MSpltrLib/fmi2TypesPlatform.h, Logical/Programs/CNC_Programs/InitiationandHoming, Logical/Programs/CNC_Programs/ManualContr/Types.typ, Logical/Programs/CNC_Programs/ManualContr/VisuAction.st, Logical/Programs/CNC_Programs/RuchZGCode, Logical/Programs/Alarm, Logical/Programs/UsrMgmtP/Types.typ, Logical/CNC_FMUFmu2/CNC_FMULib/Constants.var, Logical/CNC_FMUFmu2/CNC_FMULib/fmi2.cpp, Logical/CNC_FMUFmu2/CNC_FMULib/fmi2Functions.h, Logical/CNC_FMUFmu2/CNC_FMULib/fmi2FunctionTypes.h, Logical/CNC_FMUFmu2/CNC_FMULib/fmi2TypesPlatform.h, Logical/CNC_FMUFmu2/CNC_FMULib/CNC_FMU/fmuTemplate.h, Logical/CNC_FMUFmu2/CNC_FMUPrg/Exit.c, Logical/CNC_FMUFmu2/CNC_FMUPrg/Types.typ, Logical/live_drawing/live_draw/Types.typ, Logical/live_drawing/svgArray.var, Logical/Sources/live_drawing/svg_to_gcode
